Omron CX-Programmer project 新工程 (CX-Programmer 5.00)

# PLC 新PLC1: CQM1 CPU41

## Global symbols (name address type ; comment)
0.00 BOOL  ; 输送线全线启动
0.01 BOOL  ; 日运行停止
0.10 BOOL  ; 接触器KM1辅助触点
0.11 BOOL  ; 接触器KM2辅助触点
0.12 BOOL  ; 自动
0.13 BOOL  ; 手动
0.14 BOOL  ; 工位前占位
0.15 BOOL  ; 工位占位
100.00 BOOL  ; 输送电机M01-04接触器
100.01 BOOL  ; 输送电机M05-08接触器
100.02 BOOL  ; 输送电机M11-15接触器
100.05 BOOL  ; 输送电机M09接触器
100.06 BOOL  ; 输送电机M10接触器正转
100.07 BOOL  ; 输送电机M09接触器反转
100.10 BOOL  ; 1#密封试验开始
100.11 BOOL  ; 打号开始（接打号机）
100.12 BOOL  ; 输送线运行
101.03 BOOL  ; 自动指示灯
101.04 BOOL  ; 原位指示灯
101.05 BOOL  ; 自动指示灯
101.06 BOOL  ; 原位指示灯
101.07 BOOL  ; 自动指示灯
101.08 BOOL  ; 原位指示灯
103.00 BOOL  ; 工位前停止器
103.01 BOOL  ; 工位停止器
103.02 BOOL  ; 举升缸上升
103.03 BOOL  ; 上密封缸下降
103.04 BOOL  ; 上密封缸上升
103.05 BOOL  ; 左密封缸前进
103.06 BOOL  ; 左密封缸后退
103.07 BOOL  ; 排气孔密封缸前进
103.08 BOOL  ; 排气孔密封缸后退
103.10 BOOL  ; 2#密封试验开始
103.11 BOOL  ; 2#密封试验复位
103.12 BOOL  ; 举升缸下降
103.13 BOOL  ; 工位停止器
103.14 BOOL  ; 举升缸上升
103.15 BOOL  ; 上密封缸下降
104.00 BOOL  ; 上密封缸上升
104.01 BOOL  ; 左密封缸前进
104.02 BOOL  ; 左密封缸后退
104.03 BOOL  ; 排气孔密封缸前进
104.04 BOOL  ; 排气孔密封缸后退
104.06 BOOL  ; 工位停止器
104.07 BOOL  ; 举升缸上升
104.08 BOOL  ; 工位停止器（打号）
104.09 BOOL  ; 举升缸上升（打号）
104.10 BOOL  ; 举升缸下降（打号）
104.11 BOOL  ; 举升缸下降
104.12 BOOL  ; 举升缸下降
104.13 BOOL  ; 工位前停止器
150.02 BOOL  ; 输送线运行
160.00 BOOL  ; 自动
160.01 BOOL  ; 手动
160.03 BOOL  ; 密封机原状态
160.05 BOOL  ; 试验确认
160.07 BOOL  ; 试验不合格
160.08 BOOL  ; 试验合格
160.10 BOOL  ; 检测无工件确认
161.00 BOOL  ; 自动
161.01 BOOL  ; 手动
161.03 BOOL  ; 密封机原状态
161.05 BOOL  ; 试验确认
161.07 BOOL  ; 试验不合格
161.08 BOOL  ; 试验合格
161.10 BOOL  ; 检测无工件确认
162.00 BOOL  ; 工位前停止器
162.01 BOOL  ; 举升缸上升
162.02 BOOL  ; 举升缸下降
162.03 BOOL  ; 上密封缸下降
162.04 BOOL  ; 上密封缸上升
162.05 BOOL  ; 左密封缸前进
162.06 BOOL  ; 左密封缸后退
162.07 BOOL  ; 排气孔密封缸前进
162.08 BOOL  ; 排气孔密封缸后退
162.09 BOOL  ; 工位停止器
162.11 BOOL  ; 密封试验开始
162.14 BOOL  ; 使162.11失电
163.00 BOOL  ; 工位前停止器
163.01 BOOL  ; 举升缸上升
163.02 BOOL  ; 举升缸下降
163.03 BOOL  ; 上密封缸下降
163.04 BOOL  ; 上密封缸上升
163.05 BOOL  ; 左密封缸前进
163.06 BOOL  ; 左密封缸后退
163.07 BOOL  ; 排气孔密封缸前进
163.08 BOOL  ; 排气孔密封缸后退
163.09 BOOL  ; 工位停止器
163.11 BOOL  ; 密封试验开始
163.14 BOOL  ; 使163.11失电
170.00 BOOL  ; 自动
170.01 BOOL  ; 手动
170.03 BOOL  ; 举升缸下位
170.04 BOOL  ; 举升缸下位（打号）
172.01 BOOL  ; 举升缸上升
172.02 BOOL  ; 举升缸下降
172.05 BOOL  ; 电机M10正转
172.06 BOOL  ; 电机M09反转
172.08 BOOL  ; 工位停止器
172.10 BOOL  ; 举升缸上升（打号）
172.11 BOOL  ; 举升缸下降（打号）
172.12 BOOL  ; 工位停止器（打号）
172.13 BOOL  ; 打号开始
1.01 BOOL  ; 有无工件检测
1.02 BOOL  ; 变速箱类型检测
1.04 BOOL  ; 举升缸下位
1.05 BOOL  ; 举升缸上位
1.06 BOOL  ; 上密封缸上位
1.07 BOOL  ; 上密封缸下位
1.08 BOOL  ; 左密封缸后位
1.09 BOOL  ; 左密封缸前位
1.12 BOOL  ; 排气孔密封缸后位
1.13 BOOL  ; 排气孔密封缸前位
1.15 BOOL  ; 品种选择
2.00 BOOL  ; 试验合格
2.01 BOOL  ; 试验不合格
2.02 BOOL  ; 工件放行确认
2.04 BOOL  ; 举升缸上升
2.05 BOOL  ; 举升缸下降
2.06 BOOL  ; 上密封缸下降
2.07 BOOL  ; 上密封缸上升
2.08 BOOL  ; 左密封缸向前
2.09 BOOL  ; 左密封缸向后
2.10 BOOL  ; 排气孔密封缸向前
2.11 BOOL  ; 排气孔密封缸向后
2.12 BOOL  ; 标记缸动作
2.13 BOOL  ; 工位前停止器下
2.14 BOOL  ; 工位停止器下
2.15 BOOL  ; 信号灯测试
3.00 BOOL  ; 工件进维修段确认
3.01 BOOL  ; 自动
3.02 BOOL  ; 手动
3.03 BOOL  ; 工位占位
3.04 BOOL  ; 有无工件检测
3.05 BOOL  ; 举升缸下位
3.06 BOOL  ; 举升缸上位
3.07 BOOL  ; 上密封缸上位
3.08 BOOL  ; 上密封缸下位
3.09 BOOL  ; 左密封缸后位
3.10 BOOL  ; 左密封缸前位
3.11 BOOL  ; 排气孔密封缸后位
3.12 BOOL  ; 排气孔密封缸前位
3.13 BOOL  ; 工位前占位
3.14 BOOL  ; 试验合格
3.15 BOOL  ; 试验不合格
4.01 BOOL  ; 举升缸上升
4.02 BOOL  ; 举升缸下降
4.03 BOOL  ; 上密封缸下降
4.04 BOOL  ; 上密封缸上升
4.05 BOOL  ; 左密封缸向前
4.06 BOOL  ; 左密封缸向后
4.07 BOOL  ; 排气孔密封缸向前
4.08 BOOL  ; 排气孔密封缸向后
4.09 BOOL  ; 工位停止器下
4.10 BOOL  ; 信号灯测试
4.11 BOOL  ; 工件放行确认
4.12 BOOL  ; 工位前停止器下
4.13 BOOL  ; 预留（暂未用）
4.14 BOOL  ; 自动
4.15 BOOL  ; 手动
5.00 BOOL  ; 工位托盘占位
5.01 BOOL  ; 举升缸下位
5.02 BOOL  ; 举升缸上位
5.03 BOOL  ; 转移前到位
5.04 BOOL  ; 转移后到位
5.07 BOOL  ; 工位托盘占位（打号）
5.08 BOOL  ; 托盘满位（打号）
5.09 BOOL  ; 举升缸下位（打号）
5.10 BOOL  ; 举升缸上位（打号）
5.11 BOOL  ; 打号完毕（打号）
5.14 BOOL  ; 举升缸上升
5.15 BOOL  ; 举升缸下降
6.00 BOOL  ; 转移向前（+打号）
6.01 BOOL  ; 转移向后（+打号）
6.02 BOOL  ; 维修段放行（+打号）
6.03 BOOL  ; 出维修段确认（+打号）
6.04 BOOL  ; 打号工位举升（+打号）
6.05 BOOL  ; 打号工位下降（+打号）
6.06 BOOL  ; 打号工位放行（+打号）
6.07 BOOL  ; 信号灯测试（+打号）

## Program 新程序1 (no task)

### Section 段1_启动

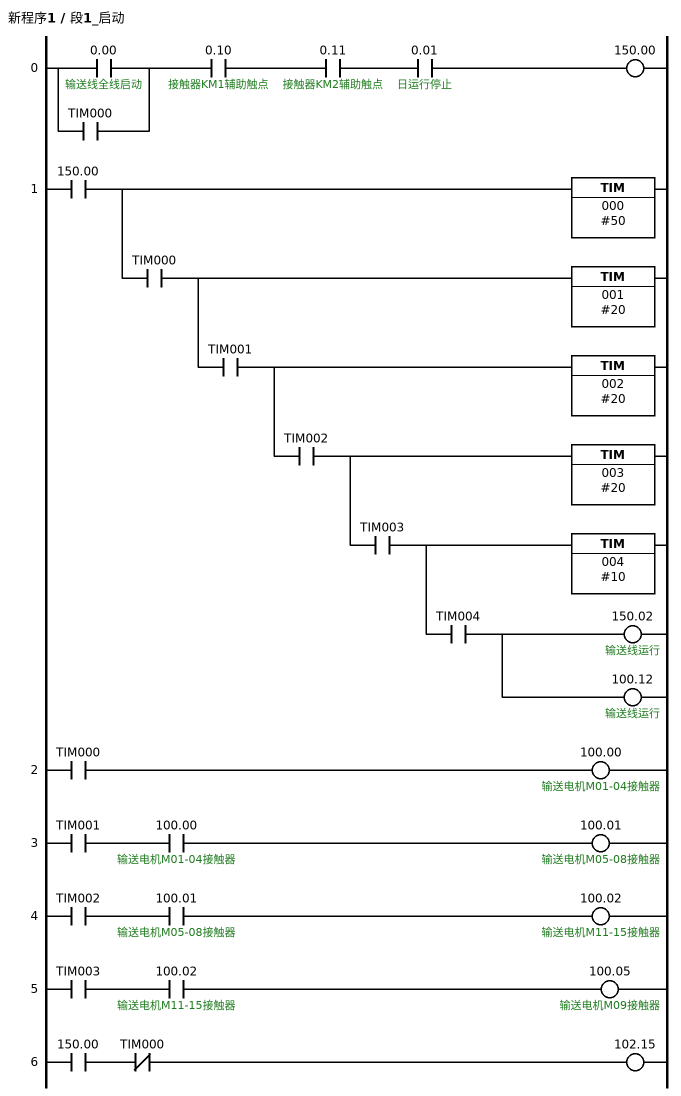
; rung 0
LD 0.00  ; 输送线全线启动
OR TIM000
AND 0.10  ; 接触器KM1辅助触点
AND 0.11  ; 接触器KM2辅助触点
AND 0.01  ; 日运行停止
OUT 150.00
; rung 1
LD 150.00
TIM 000 #50
AND TIM000
TIM 001 #20
AND TIM001
TIM 002 #20
AND TIM002
TIM 003 #20
AND TIM003
TIM 004 #10
AND TIM004
OUT 150.02  ; 输送线运行
OUT 100.12  ; 输送线运行
; rung 2
LD TIM000
OUT 100.00  ; 输送电机M01-04接触器
; rung 3
LD TIM001
AND 100.00  ; 输送电机M01-04接触器
OUT 100.01  ; 输送电机M05-08接触器
; rung 4
LD TIM002
AND 100.01  ; 输送电机M05-08接触器
OUT 100.02  ; 输送电机M11-15接触器
; rung 5
LD TIM003
AND 100.02  ; 输送电机M11-15接触器
OUT 100.05  ; 输送电机M09接触器
; rung 6
LD 150.00
ANDNOT TIM000
OUT 102.15

### Section 段2_试验机1

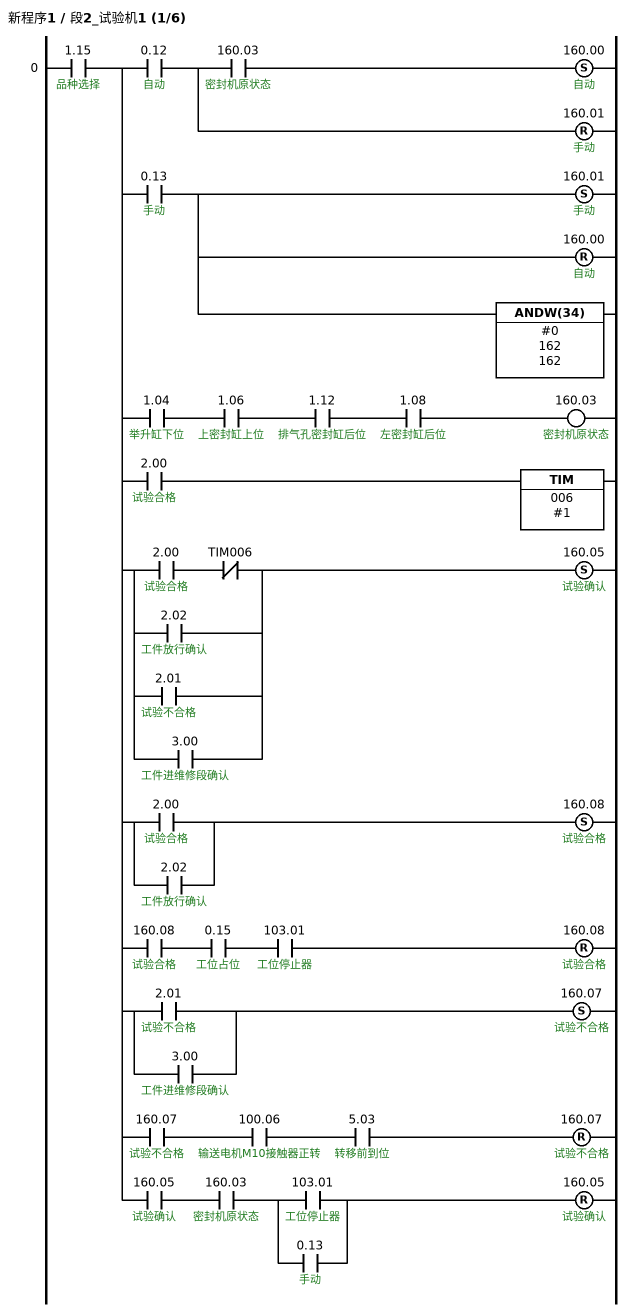
; rung 0
LD 1.15  ; 品种选择
OUT TR0
AND 0.12  ; 自动
OUT TR1
AND 160.03  ; 密封机原状态
SET 160.00  ; 自动
LD TR1
RSET 160.01  ; 手动
LD TR0
AND 0.13  ; 手动
SET 160.01  ; 手动
RSET 160.00  ; 自动
ANDW(34) #0 162 162
LD TR0
AND 1.04  ; 举升缸下位
AND 1.06  ; 上密封缸上位
AND 1.12  ; 排气孔密封缸后位
AND 1.08  ; 左密封缸后位
OUT 160.03  ; 密封机原状态
LD TR0
AND 2.00  ; 试验合格
TIM 006 #1
LD TR0
LD 2.00  ; 试验合格
ANDNOT TIM006
OR 2.02  ; 工件放行确认
OR 2.01  ; 试验不合格
OR 3.00  ; 工件进维修段确认
ANDLD
SET 160.05  ; 试验确认
LD TR0
LD 2.00  ; 试验合格
OR 2.02  ; 工件放行确认
ANDLD
SET 160.08  ; 试验合格
LD TR0
AND 160.08  ; 试验合格
AND 0.15  ; 工位占位
AND 103.01  ; 工位停止器
RSET 160.08  ; 试验合格
LD TR0
LD 2.01  ; 试验不合格
OR 3.00  ; 工件进维修段确认
ANDLD
SET 160.07  ; 试验不合格
LD TR0
AND 160.07  ; 试验不合格
AND 100.06  ; 输送电机M10接触器正转
AND 5.03  ; 转移前到位
RSET 160.07  ; 试验不合格
LD TR0
AND 160.05  ; 试验确认
AND 160.03  ; 密封机原状态
LD 103.01  ; 工位停止器
OR 0.13  ; 手动
ANDLD
RSET 160.05  ; 试验确认

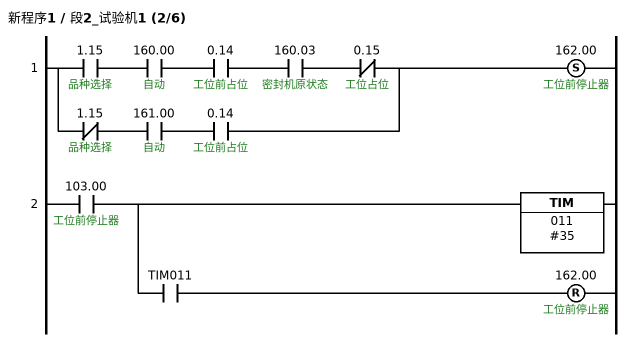
; rung 1
LD 1.15  ; 品种选择
AND 160.00  ; 自动
AND 0.14  ; 工位前占位
AND 160.03  ; 密封机原状态
ANDNOT 0.15  ; 工位占位
LDNOT 1.15  ; 品种选择
AND 161.00  ; 自动
AND 0.14  ; 工位前占位
ORLD
SET 162.00  ; 工位前停止器
; rung 2
LD 103.00  ; 工位前停止器
TIM 011 #35
AND TIM011
RSET 162.00  ; 工位前停止器

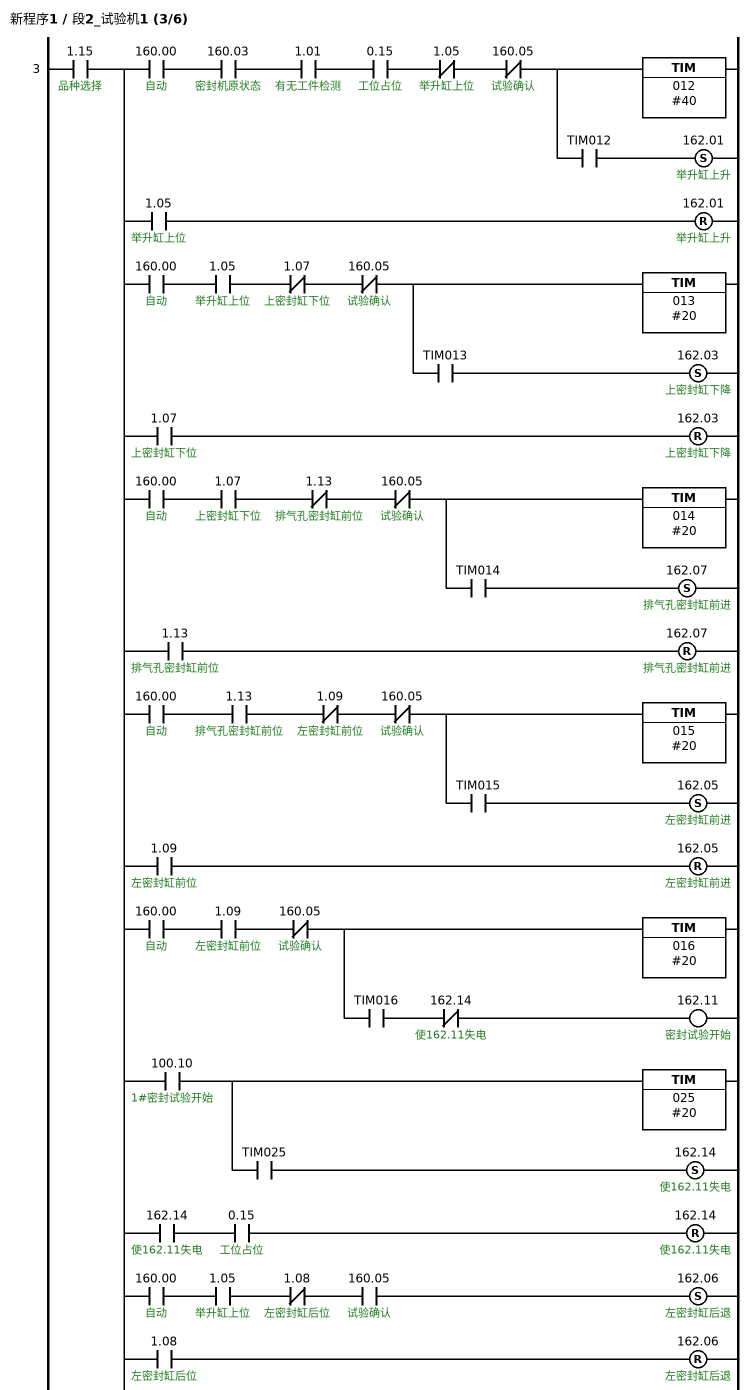

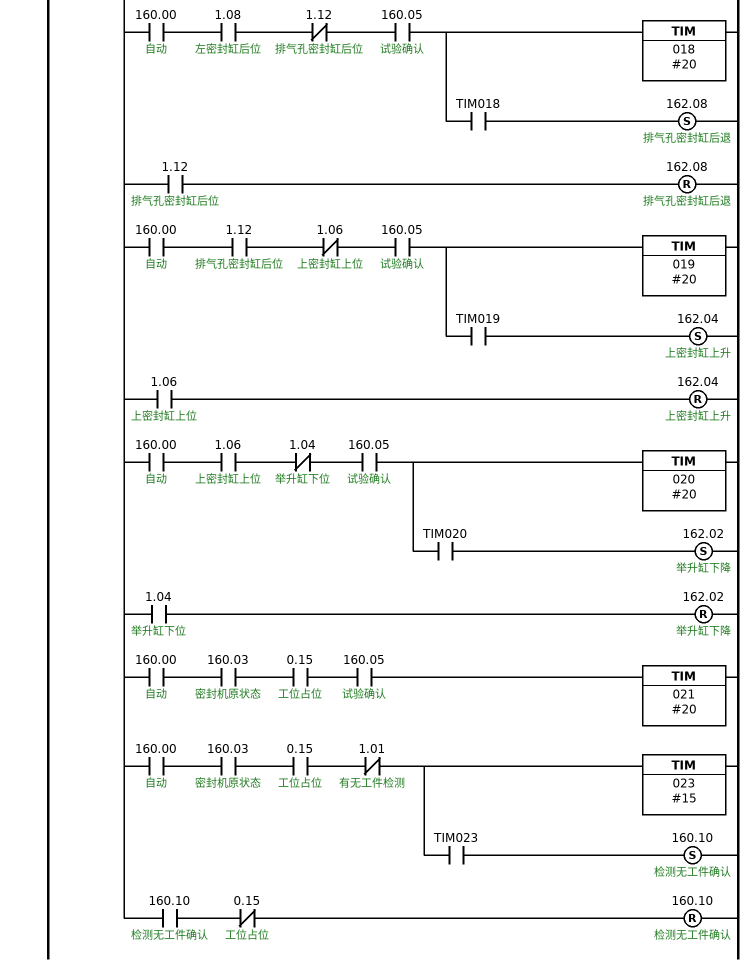
; rung 3
LD 1.15  ; 品种选择
OUT TR0
AND 160.00  ; 自动
AND 160.03  ; 密封机原状态
AND 1.01  ; 有无工件检测
AND 0.15  ; 工位占位
ANDNOT 1.05  ; 举升缸上位
ANDNOT 160.05  ; 试验确认
TIM 012 #40
AND TIM012
SET 162.01  ; 举升缸上升
LD TR0
AND 1.05  ; 举升缸上位
RSET 162.01  ; 举升缸上升
LD TR0
AND 160.00  ; 自动
AND 1.05  ; 举升缸上位
ANDNOT 1.07  ; 上密封缸下位
ANDNOT 160.05  ; 试验确认
TIM 013 #20
AND TIM013
SET 162.03  ; 上密封缸下降
LD TR0
AND 1.07  ; 上密封缸下位
RSET 162.03  ; 上密封缸下降
LD TR0
AND 160.00  ; 自动
AND 1.07  ; 上密封缸下位
ANDNOT 1.13  ; 排气孔密封缸前位
ANDNOT 160.05  ; 试验确认
TIM 014 #20
AND TIM014
SET 162.07  ; 排气孔密封缸前进
LD TR0
AND 1.13  ; 排气孔密封缸前位
RSET 162.07  ; 排气孔密封缸前进
LD TR0
AND 160.00  ; 自动
AND 1.13  ; 排气孔密封缸前位
ANDNOT 1.09  ; 左密封缸前位
ANDNOT 160.05  ; 试验确认
TIM 015 #20
AND TIM015
SET 162.05  ; 左密封缸前进
LD TR0
AND 1.09  ; 左密封缸前位
RSET 162.05  ; 左密封缸前进
LD TR0
AND 160.00  ; 自动
AND 1.09  ; 左密封缸前位
ANDNOT 160.05  ; 试验确认
TIM 016 #20
AND TIM016
ANDNOT 162.14  ; 使162.11失电
OUT 162.11  ; 密封试验开始
LD TR0
AND 100.10  ; 1#密封试验开始
TIM 025 #20
AND TIM025
SET 162.14  ; 使162.11失电
LD TR0
AND 162.14  ; 使162.11失电
AND 0.15  ; 工位占位
RSET 162.14  ; 使162.11失电
LD TR0
AND 160.00  ; 自动
AND 1.05  ; 举升缸上位
ANDNOT 1.08  ; 左密封缸后位
AND 160.05  ; 试验确认
SET 162.06  ; 左密封缸后退
LD TR0
AND 1.08  ; 左密封缸后位
RSET 162.06  ; 左密封缸后退
LD TR0
AND 160.00  ; 自动
AND 1.08  ; 左密封缸后位
ANDNOT 1.12  ; 排气孔密封缸后位
AND 160.05  ; 试验确认
TIM 018 #20
AND TIM018
SET 162.08  ; 排气孔密封缸后退
LD TR0
AND 1.12  ; 排气孔密封缸后位
RSET 162.08  ; 排气孔密封缸后退
LD TR0
AND 160.00  ; 自动
AND 1.12  ; 排气孔密封缸后位
ANDNOT 1.06  ; 上密封缸上位
AND 160.05  ; 试验确认
TIM 019 #20
AND TIM019
SET 162.04  ; 上密封缸上升
LD TR0
AND 1.06  ; 上密封缸上位
RSET 162.04  ; 上密封缸上升
LD TR0
AND 160.00  ; 自动
AND 1.06  ; 上密封缸上位
ANDNOT 1.04  ; 举升缸下位
AND 160.05  ; 试验确认
TIM 020 #20
AND TIM020
SET 162.02  ; 举升缸下降
LD TR0
AND 1.04  ; 举升缸下位
RSET 162.02  ; 举升缸下降
LD TR0
AND 160.00  ; 自动
AND 160.03  ; 密封机原状态
AND 0.15  ; 工位占位
AND 160.05  ; 试验确认
TIM 021 #20
LD TR0
AND 160.00  ; 自动
AND 160.03  ; 密封机原状态
AND 0.15  ; 工位占位
ANDNOT 1.01  ; 有无工件检测
TIM 023 #15
AND TIM023
SET 160.10  ; 检测无工件确认
LD TR0
AND 160.10  ; 检测无工件确认
ANDNOT 0.15  ; 工位占位
RSET 160.10  ; 检测无工件确认

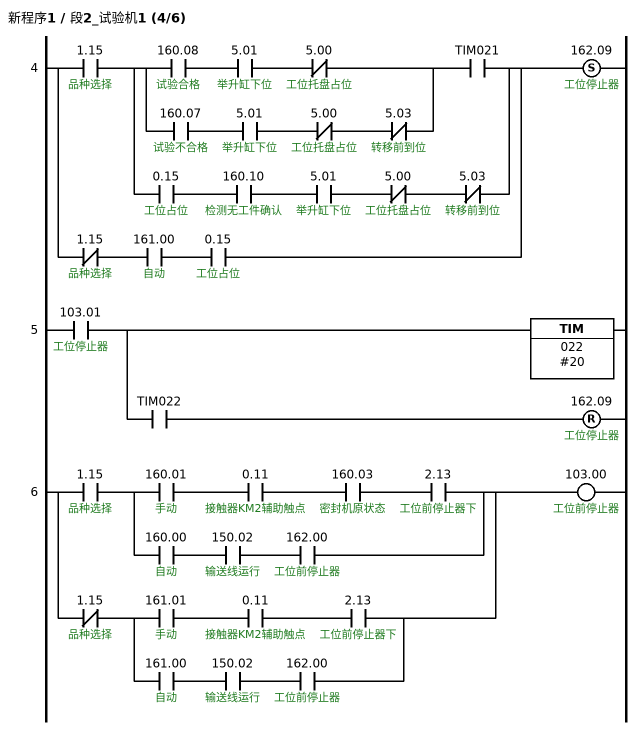
; rung 4
LD 1.15  ; 品种选择
LD 160.08  ; 试验合格
AND 5.01  ; 举升缸下位
ANDNOT 5.00  ; 工位托盘占位
LD 160.07  ; 试验不合格
AND 5.01  ; 举升缸下位
ANDNOT 5.00  ; 工位托盘占位
ANDNOT 5.03  ; 转移前到位
ORLD
AND TIM021
LD 0.15  ; 工位占位
AND 160.10  ; 检测无工件确认
AND 5.01  ; 举升缸下位
ANDNOT 5.00  ; 工位托盘占位
ANDNOT 5.03  ; 转移前到位
ORLD
ANDLD
LDNOT 1.15  ; 品种选择
AND 161.00  ; 自动
AND 0.15  ; 工位占位
ORLD
SET 162.09  ; 工位停止器
; rung 5
LD 103.01  ; 工位停止器
TIM 022 #20
AND TIM022
RSET 162.09  ; 工位停止器
; rung 6
LD 1.15  ; 品种选择
LD 160.01  ; 手动
AND 0.11  ; 接触器KM2辅助触点
AND 160.03  ; 密封机原状态
AND 2.13  ; 工位前停止器下
LD 160.00  ; 自动
AND 150.02  ; 输送线运行
AND 162.00  ; 工位前停止器
ORLD
ANDLD
LDNOT 1.15  ; 品种选择
LD 161.01  ; 手动
AND 0.11  ; 接触器KM2辅助触点
AND 2.13  ; 工位前停止器下
LD 161.00  ; 自动
AND 150.02  ; 输送线运行
AND 162.00  ; 工位前停止器
ORLD
ANDLD
ORLD
OUT 103.00  ; 工位前停止器

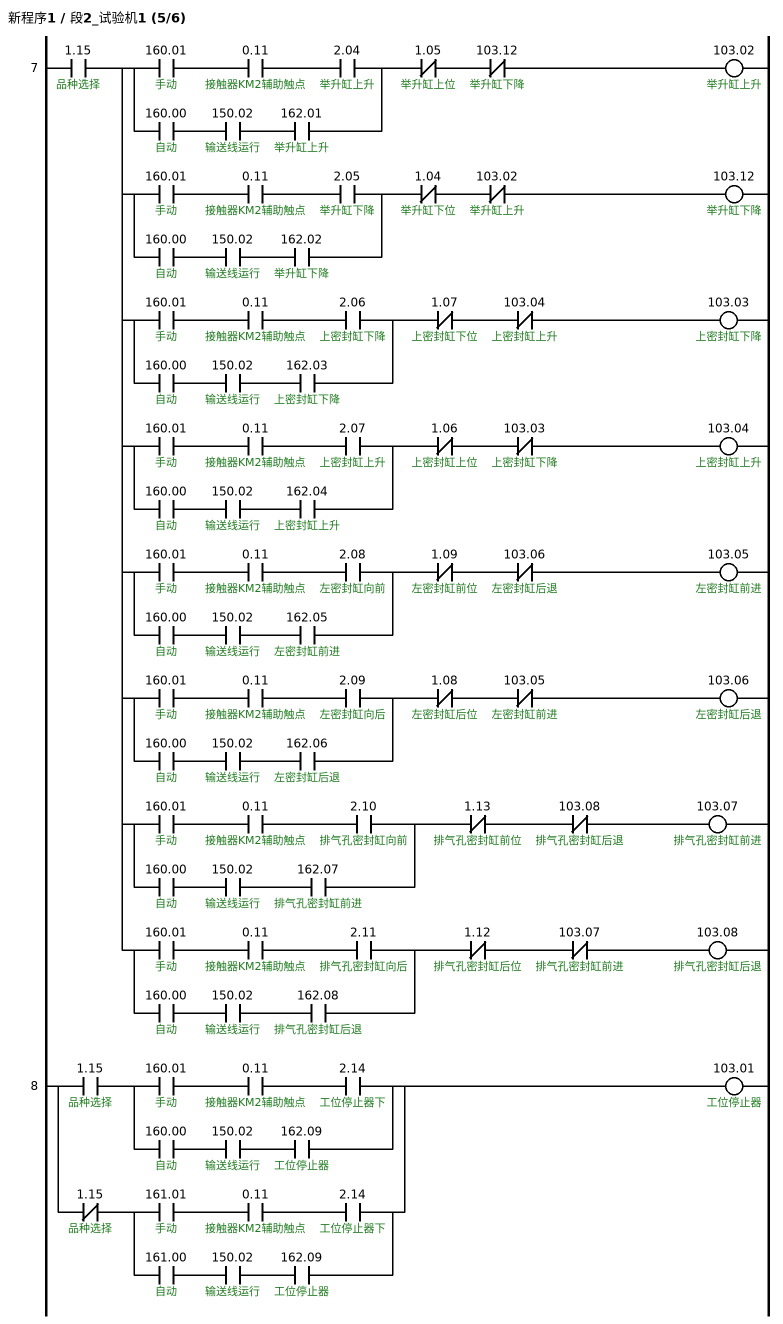
; rung 7
LD 1.15  ; 品种选择
OUT TR0
LD 160.01  ; 手动
AND 0.11  ; 接触器KM2辅助触点
AND 2.04  ; 举升缸上升
LD 160.00  ; 自动
AND 150.02  ; 输送线运行
AND 162.01  ; 举升缸上升
ORLD
ANDLD
ANDNOT 1.05  ; 举升缸上位
ANDNOT 103.12  ; 举升缸下降
OUT 103.02  ; 举升缸上升
LD TR0
LD 160.01  ; 手动
AND 0.11  ; 接触器KM2辅助触点
AND 2.05  ; 举升缸下降
LD 160.00  ; 自动
AND 150.02  ; 输送线运行
AND 162.02  ; 举升缸下降
ORLD
ANDLD
ANDNOT 1.04  ; 举升缸下位
ANDNOT 103.02  ; 举升缸上升
OUT 103.12  ; 举升缸下降
LD TR0
LD 160.01  ; 手动
AND 0.11  ; 接触器KM2辅助触点
AND 2.06  ; 上密封缸下降
LD 160.00  ; 自动
AND 150.02  ; 输送线运行
AND 162.03  ; 上密封缸下降
ORLD
ANDLD
ANDNOT 1.07  ; 上密封缸下位
ANDNOT 103.04  ; 上密封缸上升
OUT 103.03  ; 上密封缸下降
LD TR0
LD 160.01  ; 手动
AND 0.11  ; 接触器KM2辅助触点
AND 2.07  ; 上密封缸上升
LD 160.00  ; 自动
AND 150.02  ; 输送线运行
AND 162.04  ; 上密封缸上升
ORLD
ANDLD
ANDNOT 1.06  ; 上密封缸上位
ANDNOT 103.03  ; 上密封缸下降
OUT 103.04  ; 上密封缸上升
LD TR0
LD 160.01  ; 手动
AND 0.11  ; 接触器KM2辅助触点
AND 2.08  ; 左密封缸向前
LD 160.00  ; 自动
AND 150.02  ; 输送线运行
AND 162.05  ; 左密封缸前进
ORLD
ANDLD
ANDNOT 1.09  ; 左密封缸前位
ANDNOT 103.06  ; 左密封缸后退
OUT 103.05  ; 左密封缸前进
LD TR0
LD 160.01  ; 手动
AND 0.11  ; 接触器KM2辅助触点
AND 2.09  ; 左密封缸向后
LD 160.00  ; 自动
AND 150.02  ; 输送线运行
AND 162.06  ; 左密封缸后退
ORLD
ANDLD
ANDNOT 1.08  ; 左密封缸后位
ANDNOT 103.05  ; 左密封缸前进
OUT 103.06  ; 左密封缸后退
LD TR0
LD 160.01  ; 手动
AND 0.11  ; 接触器KM2辅助触点
AND 2.10  ; 排气孔密封缸向前
LD 160.00  ; 自动
AND 150.02  ; 输送线运行
AND 162.07  ; 排气孔密封缸前进
ORLD
ANDLD
ANDNOT 1.13  ; 排气孔密封缸前位
ANDNOT 103.08  ; 排气孔密封缸后退
OUT 103.07  ; 排气孔密封缸前进
LD TR0
LD 160.01  ; 手动
AND 0.11  ; 接触器KM2辅助触点
AND 2.11  ; 排气孔密封缸向后
LD 160.00  ; 自动
AND 150.02  ; 输送线运行
AND 162.08  ; 排气孔密封缸后退
ORLD
ANDLD
ANDNOT 1.12  ; 排气孔密封缸后位
ANDNOT 103.07  ; 排气孔密封缸前进
OUT 103.08  ; 排气孔密封缸后退
; rung 8
LD 1.15  ; 品种选择
LD 160.01  ; 手动
AND 0.11  ; 接触器KM2辅助触点
AND 2.14  ; 工位停止器下
LD 160.00  ; 自动
AND 150.02  ; 输送线运行
AND 162.09  ; 工位停止器
ORLD
ANDLD
LDNOT 1.15  ; 品种选择
LD 161.01  ; 手动
AND 0.11  ; 接触器KM2辅助触点
AND 2.14  ; 工位停止器下
LD 161.00  ; 自动
AND 150.02  ; 输送线运行
AND 162.09  ; 工位停止器
ORLD
ANDLD
ORLD
OUT 103.01  ; 工位停止器

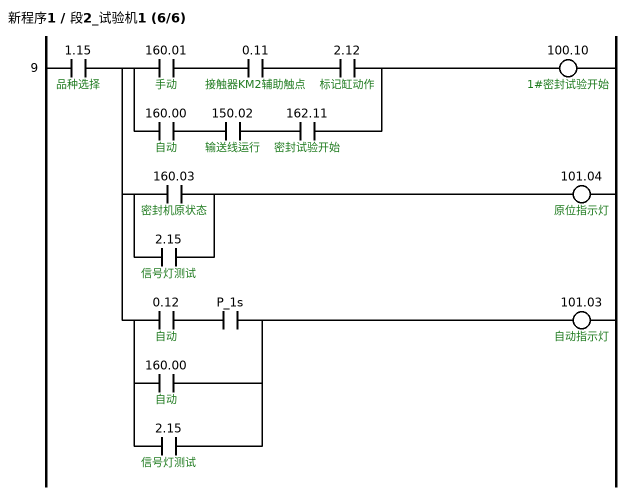
; rung 9
LD 1.15  ; 品种选择
OUT TR0
LD 160.01  ; 手动
AND 0.11  ; 接触器KM2辅助触点
AND 2.12  ; 标记缸动作
LD 160.00  ; 自动
AND 150.02  ; 输送线运行
AND 162.11  ; 密封试验开始
ORLD
ANDLD
OUT 100.10  ; 1#密封试验开始
LD TR0
LD 160.03  ; 密封机原状态
OR 2.15  ; 信号灯测试
ANDLD
OUT 101.04  ; 原位指示灯
LD TR0
LD 0.12  ; 自动
AND P_1s
OR 160.00  ; 自动
OR 2.15  ; 信号灯测试
ANDLD
OUT 101.03  ; 自动指示灯

### Section 段3_试验机2

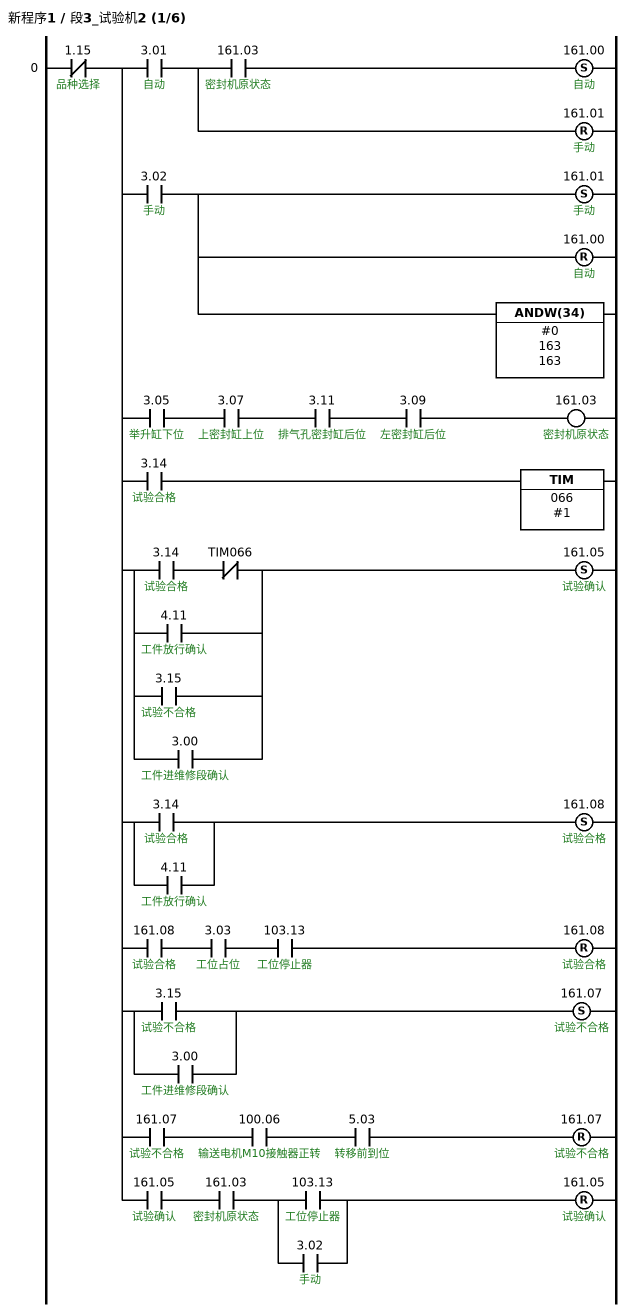
; rung 0
LDNOT 1.15  ; 品种选择
OUT TR0
AND 3.01  ; 自动
OUT TR1
AND 161.03  ; 密封机原状态
SET 161.00  ; 自动
LD TR1
RSET 161.01  ; 手动
LD TR0
AND 3.02  ; 手动
SET 161.01  ; 手动
RSET 161.00  ; 自动
ANDW(34) #0 163 163
LD TR0
AND 3.05  ; 举升缸下位
AND 3.07  ; 上密封缸上位
AND 3.11  ; 排气孔密封缸后位
AND 3.09  ; 左密封缸后位
OUT 161.03  ; 密封机原状态
LD TR0
AND 3.14  ; 试验合格
TIM 066 #1
LD TR0
LD 3.14  ; 试验合格
ANDNOT TIM066
OR 4.11  ; 工件放行确认
OR 3.15  ; 试验不合格
OR 3.00  ; 工件进维修段确认
ANDLD
SET 161.05  ; 试验确认
LD TR0
LD 3.14  ; 试验合格
OR 4.11  ; 工件放行确认
ANDLD
SET 161.08  ; 试验合格
LD TR0
AND 161.08  ; 试验合格
AND 3.03  ; 工位占位
AND 103.13  ; 工位停止器
RSET 161.08  ; 试验合格
LD TR0
LD 3.15  ; 试验不合格
OR 3.00  ; 工件进维修段确认
ANDLD
SET 161.07  ; 试验不合格
LD TR0
AND 161.07  ; 试验不合格
AND 100.06  ; 输送电机M10接触器正转
AND 5.03  ; 转移前到位
RSET 161.07  ; 试验不合格
LD TR0
AND 161.05  ; 试验确认
AND 161.03  ; 密封机原状态
LD 103.13  ; 工位停止器
OR 3.02  ; 手动
ANDLD
RSET 161.05  ; 试验确认

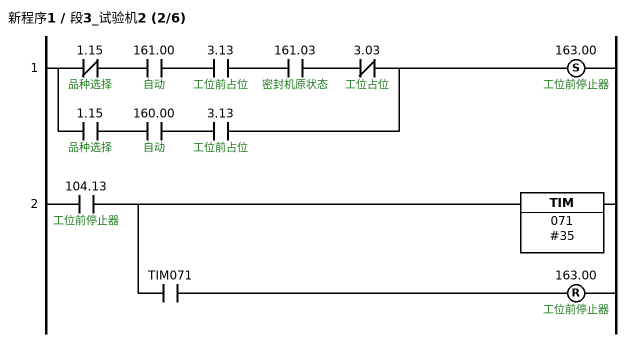
; rung 1
LDNOT 1.15  ; 品种选择
AND 161.00  ; 自动
AND 3.13  ; 工位前占位
AND 161.03  ; 密封机原状态
ANDNOT 3.03  ; 工位占位
LD 1.15  ; 品种选择
AND 160.00  ; 自动
AND 3.13  ; 工位前占位
ORLD
SET 163.00  ; 工位前停止器
; rung 2
LD 104.13  ; 工位前停止器
TIM 071 #35
AND TIM071
RSET 163.00  ; 工位前停止器

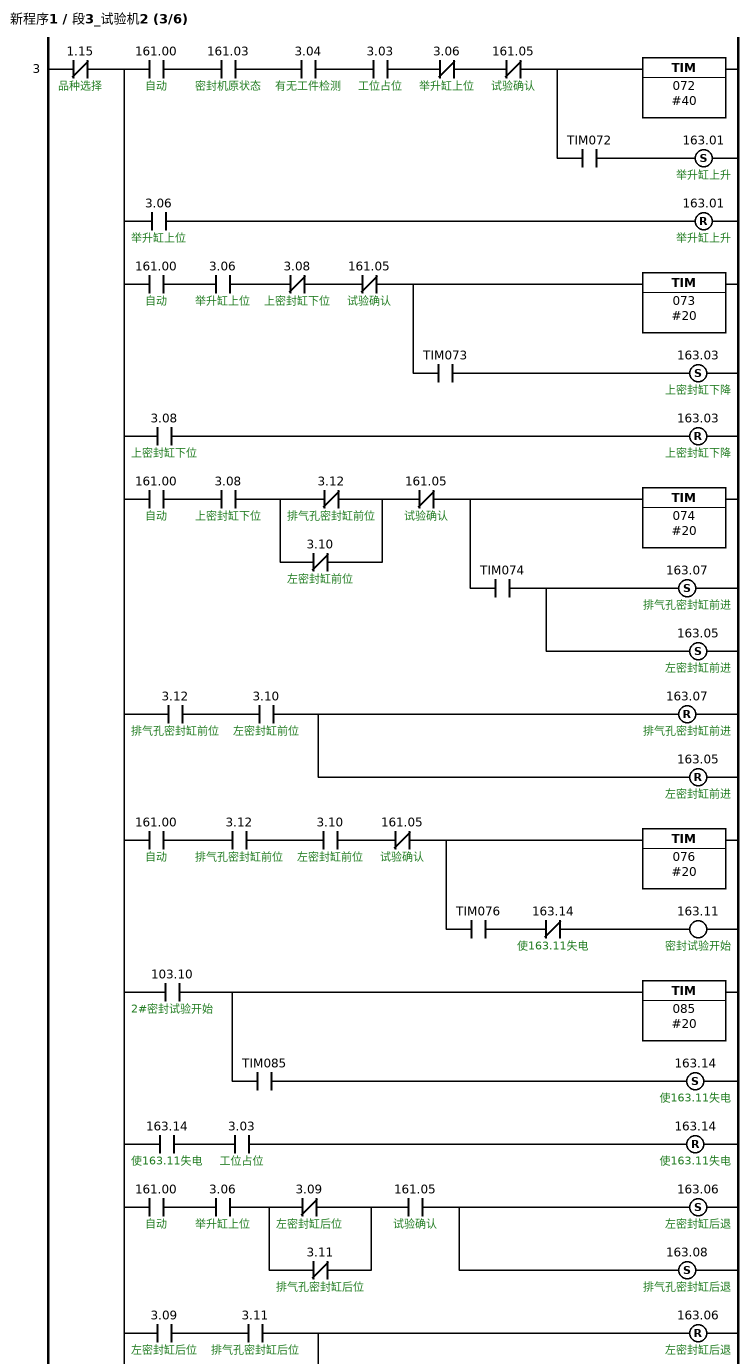

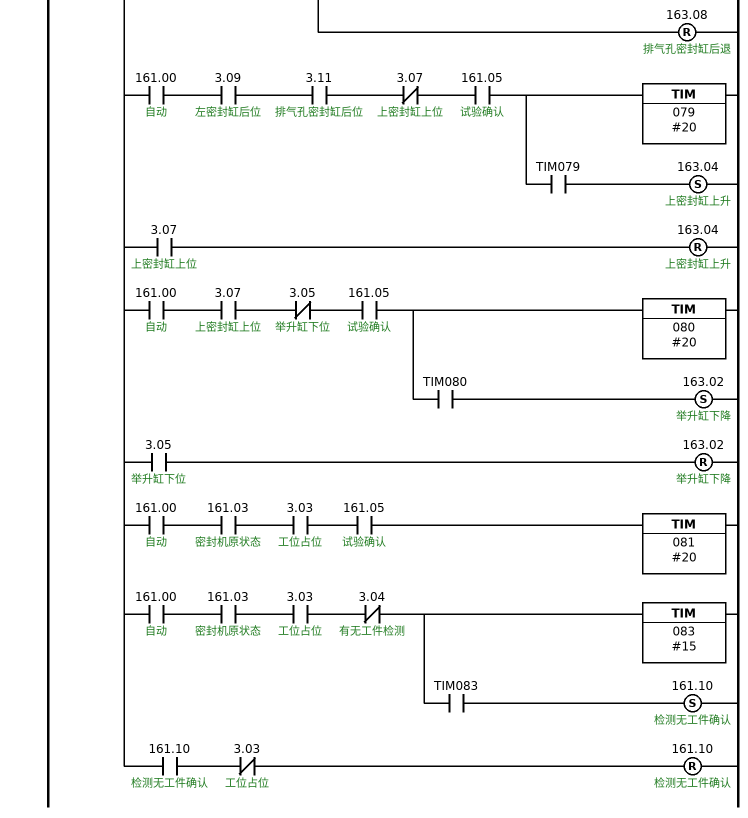
; rung 3
LDNOT 1.15  ; 品种选择
OUT TR0
AND 161.00  ; 自动
AND 161.03  ; 密封机原状态
AND 3.04  ; 有无工件检测
AND 3.03  ; 工位占位
ANDNOT 3.06  ; 举升缸上位
ANDNOT 161.05  ; 试验确认
TIM 072 #40
AND TIM072
SET 163.01  ; 举升缸上升
LD TR0
AND 3.06  ; 举升缸上位
RSET 163.01  ; 举升缸上升
LD TR0
AND 161.00  ; 自动
AND 3.06  ; 举升缸上位
ANDNOT 3.08  ; 上密封缸下位
ANDNOT 161.05  ; 试验确认
TIM 073 #20
AND TIM073
SET 163.03  ; 上密封缸下降
LD TR0
AND 3.08  ; 上密封缸下位
RSET 163.03  ; 上密封缸下降
LD TR0
AND 161.00  ; 自动
AND 3.08  ; 上密封缸下位
LDNOT 3.12  ; 排气孔密封缸前位
ORNOT 3.10  ; 左密封缸前位
ANDLD
ANDNOT 161.05  ; 试验确认
TIM 074 #20
AND TIM074
SET 163.07  ; 排气孔密封缸前进
SET 163.05  ; 左密封缸前进
LD TR0
AND 3.12  ; 排气孔密封缸前位
AND 3.10  ; 左密封缸前位
RSET 163.07  ; 排气孔密封缸前进
RSET 163.05  ; 左密封缸前进
LD TR0
AND 161.00  ; 自动
AND 3.12  ; 排气孔密封缸前位
AND 3.10  ; 左密封缸前位
ANDNOT 161.05  ; 试验确认
TIM 076 #20
AND TIM076
ANDNOT 163.14  ; 使163.11失电
OUT 163.11  ; 密封试验开始
LD TR0
AND 103.10  ; 2#密封试验开始
TIM 085 #20
AND TIM085
SET 163.14  ; 使163.11失电
LD TR0
AND 163.14  ; 使163.11失电
AND 3.03  ; 工位占位
RSET 163.14  ; 使163.11失电
LD TR0
AND 161.00  ; 自动
AND 3.06  ; 举升缸上位
LDNOT 3.09  ; 左密封缸后位
ORNOT 3.11  ; 排气孔密封缸后位
ANDLD
AND 161.05  ; 试验确认
SET 163.06  ; 左密封缸后退
SET 163.08  ; 排气孔密封缸后退
LD TR0
AND 3.09  ; 左密封缸后位
AND 3.11  ; 排气孔密封缸后位
RSET 163.06  ; 左密封缸后退
RSET 163.08  ; 排气孔密封缸后退
LD TR0
AND 161.00  ; 自动
AND 3.09  ; 左密封缸后位
AND 3.11  ; 排气孔密封缸后位
ANDNOT 3.07  ; 上密封缸上位
AND 161.05  ; 试验确认
TIM 079 #20
AND TIM079
SET 163.04  ; 上密封缸上升
LD TR0
AND 3.07  ; 上密封缸上位
RSET 163.04  ; 上密封缸上升
LD TR0
AND 161.00  ; 自动
AND 3.07  ; 上密封缸上位
ANDNOT 3.05  ; 举升缸下位
AND 161.05  ; 试验确认
TIM 080 #20
AND TIM080
SET 163.02  ; 举升缸下降
LD TR0
AND 3.05  ; 举升缸下位
RSET 163.02  ; 举升缸下降
LD TR0
AND 161.00  ; 自动
AND 161.03  ; 密封机原状态
AND 3.03  ; 工位占位
AND 161.05  ; 试验确认
TIM 081 #20
LD TR0
AND 161.00  ; 自动
AND 161.03  ; 密封机原状态
AND 3.03  ; 工位占位
ANDNOT 3.04  ; 有无工件检测
TIM 083 #15
AND TIM083
SET 161.10  ; 检测无工件确认
LD TR0
AND 161.10  ; 检测无工件确认
ANDNOT 3.03  ; 工位占位
RSET 161.10  ; 检测无工件确认

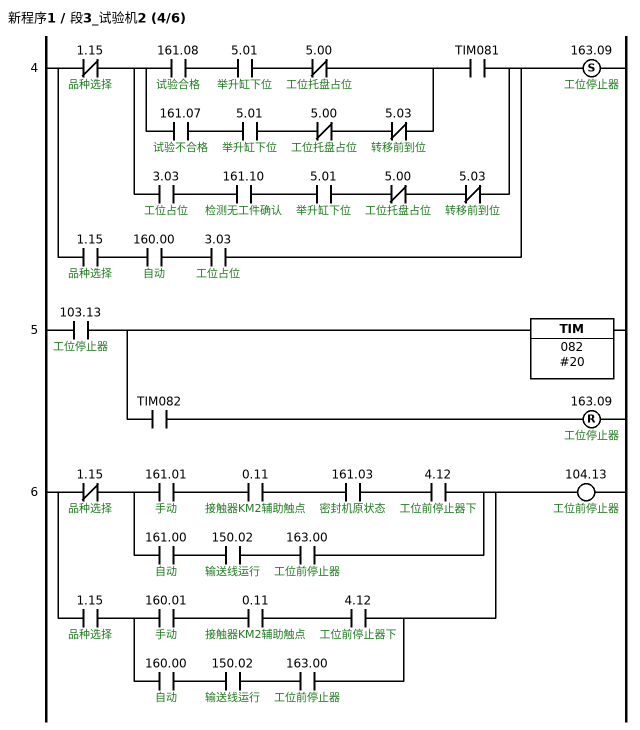
; rung 4
LDNOT 1.15  ; 品种选择
LD 161.08  ; 试验合格
AND 5.01  ; 举升缸下位
ANDNOT 5.00  ; 工位托盘占位
LD 161.07  ; 试验不合格
AND 5.01  ; 举升缸下位
ANDNOT 5.00  ; 工位托盘占位
ANDNOT 5.03  ; 转移前到位
ORLD
AND TIM081
LD 3.03  ; 工位占位
AND 161.10  ; 检测无工件确认
AND 5.01  ; 举升缸下位
ANDNOT 5.00  ; 工位托盘占位
ANDNOT 5.03  ; 转移前到位
ORLD
ANDLD
LD 1.15  ; 品种选择
AND 160.00  ; 自动
AND 3.03  ; 工位占位
ORLD
SET 163.09  ; 工位停止器
; rung 5
LD 103.13  ; 工位停止器
TIM 082 #20
AND TIM082
RSET 163.09  ; 工位停止器
; rung 6
LDNOT 1.15  ; 品种选择
LD 161.01  ; 手动
AND 0.11  ; 接触器KM2辅助触点
AND 161.03  ; 密封机原状态
AND 4.12  ; 工位前停止器下
LD 161.00  ; 自动
AND 150.02  ; 输送线运行
AND 163.00  ; 工位前停止器
ORLD
ANDLD
LD 1.15  ; 品种选择
LD 160.01  ; 手动
AND 0.11  ; 接触器KM2辅助触点
AND 4.12  ; 工位前停止器下
LD 160.00  ; 自动
AND 150.02  ; 输送线运行
AND 163.00  ; 工位前停止器
ORLD
ANDLD
ORLD
OUT 104.13  ; 工位前停止器

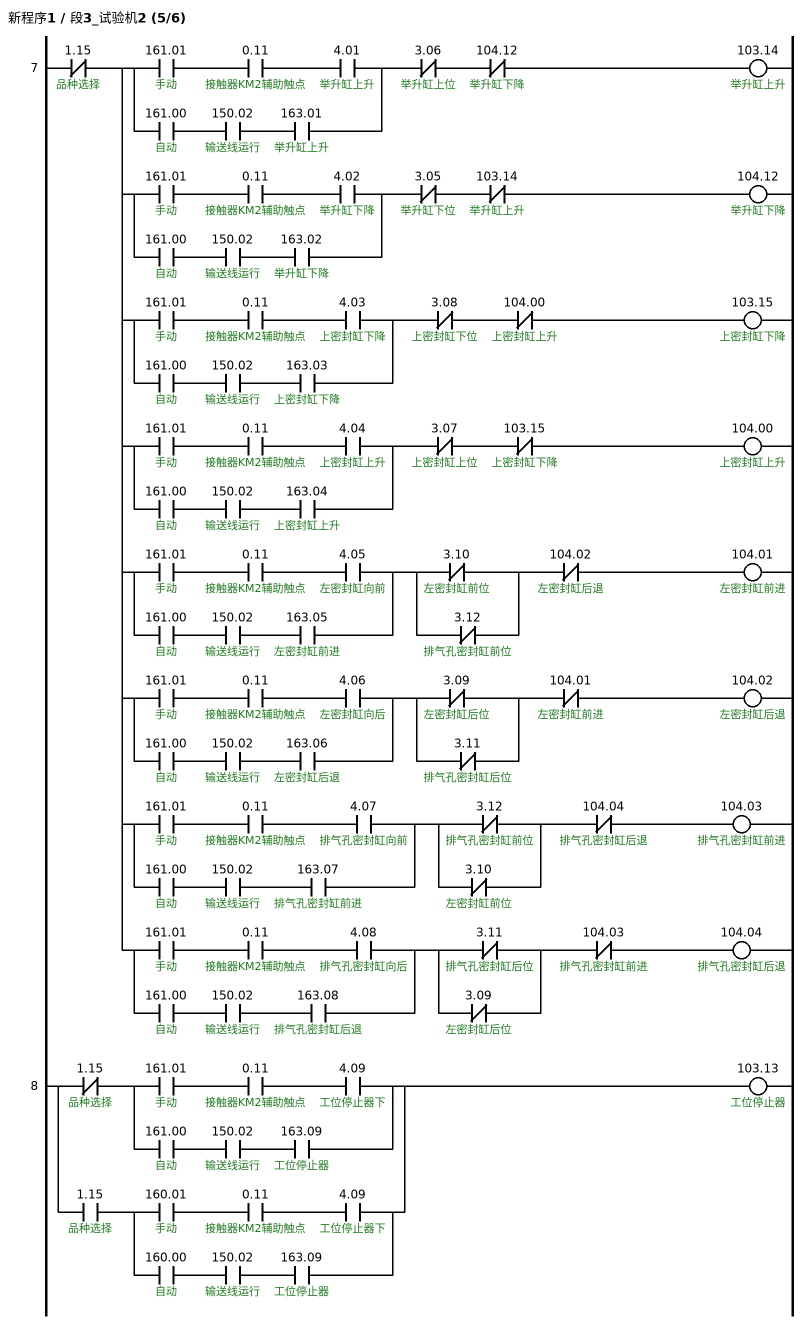
; rung 7
LDNOT 1.15  ; 品种选择
OUT TR0
LD 161.01  ; 手动
AND 0.11  ; 接触器KM2辅助触点
AND 4.01  ; 举升缸上升
LD 161.00  ; 自动
AND 150.02  ; 输送线运行
AND 163.01  ; 举升缸上升
ORLD
ANDLD
ANDNOT 3.06  ; 举升缸上位
ANDNOT 104.12  ; 举升缸下降
OUT 103.14  ; 举升缸上升
LD TR0
LD 161.01  ; 手动
AND 0.11  ; 接触器KM2辅助触点
AND 4.02  ; 举升缸下降
LD 161.00  ; 自动
AND 150.02  ; 输送线运行
AND 163.02  ; 举升缸下降
ORLD
ANDLD
ANDNOT 3.05  ; 举升缸下位
ANDNOT 103.14  ; 举升缸上升
OUT 104.12  ; 举升缸下降
LD TR0
LD 161.01  ; 手动
AND 0.11  ; 接触器KM2辅助触点
AND 4.03  ; 上密封缸下降
LD 161.00  ; 自动
AND 150.02  ; 输送线运行
AND 163.03  ; 上密封缸下降
ORLD
ANDLD
ANDNOT 3.08  ; 上密封缸下位
ANDNOT 104.00  ; 上密封缸上升
OUT 103.15  ; 上密封缸下降
LD TR0
LD 161.01  ; 手动
AND 0.11  ; 接触器KM2辅助触点
AND 4.04  ; 上密封缸上升
LD 161.00  ; 自动
AND 150.02  ; 输送线运行
AND 163.04  ; 上密封缸上升
ORLD
ANDLD
ANDNOT 3.07  ; 上密封缸上位
ANDNOT 103.15  ; 上密封缸下降
OUT 104.00  ; 上密封缸上升
LD TR0
LD 161.01  ; 手动
AND 0.11  ; 接触器KM2辅助触点
AND 4.05  ; 左密封缸向前
LD 161.00  ; 自动
AND 150.02  ; 输送线运行
AND 163.05  ; 左密封缸前进
ORLD
ANDLD
LDNOT 3.10  ; 左密封缸前位
ORNOT 3.12  ; 排气孔密封缸前位
ANDLD
ANDNOT 104.02  ; 左密封缸后退
OUT 104.01  ; 左密封缸前进
LD TR0
LD 161.01  ; 手动
AND 0.11  ; 接触器KM2辅助触点
AND 4.06  ; 左密封缸向后
LD 161.00  ; 自动
AND 150.02  ; 输送线运行
AND 163.06  ; 左密封缸后退
ORLD
ANDLD
LDNOT 3.09  ; 左密封缸后位
ORNOT 3.11  ; 排气孔密封缸后位
ANDLD
ANDNOT 104.01  ; 左密封缸前进
OUT 104.02  ; 左密封缸后退
LD TR0
LD 161.01  ; 手动
AND 0.11  ; 接触器KM2辅助触点
AND 4.07  ; 排气孔密封缸向前
LD 161.00  ; 自动
AND 150.02  ; 输送线运行
AND 163.07  ; 排气孔密封缸前进
ORLD
ANDLD
LDNOT 3.12  ; 排气孔密封缸前位
ORNOT 3.10  ; 左密封缸前位
ANDLD
ANDNOT 104.04  ; 排气孔密封缸后退
OUT 104.03  ; 排气孔密封缸前进
LD TR0
LD 161.01  ; 手动
AND 0.11  ; 接触器KM2辅助触点
AND 4.08  ; 排气孔密封缸向后
LD 161.00  ; 自动
AND 150.02  ; 输送线运行
AND 163.08  ; 排气孔密封缸后退
ORLD
ANDLD
LDNOT 3.11  ; 排气孔密封缸后位
ORNOT 3.09  ; 左密封缸后位
ANDLD
ANDNOT 104.03  ; 排气孔密封缸前进
OUT 104.04  ; 排气孔密封缸后退
; rung 8
LDNOT 1.15  ; 品种选择
LD 161.01  ; 手动
AND 0.11  ; 接触器KM2辅助触点
AND 4.09  ; 工位停止器下
LD 161.00  ; 自动
AND 150.02  ; 输送线运行
AND 163.09  ; 工位停止器
ORLD
ANDLD
LD 1.15  ; 品种选择
LD 160.01  ; 手动
AND 0.11  ; 接触器KM2辅助触点
AND 4.09  ; 工位停止器下
LD 160.00  ; 自动
AND 150.02  ; 输送线运行
AND 163.09  ; 工位停止器
ORLD
ANDLD
ORLD
OUT 103.13  ; 工位停止器

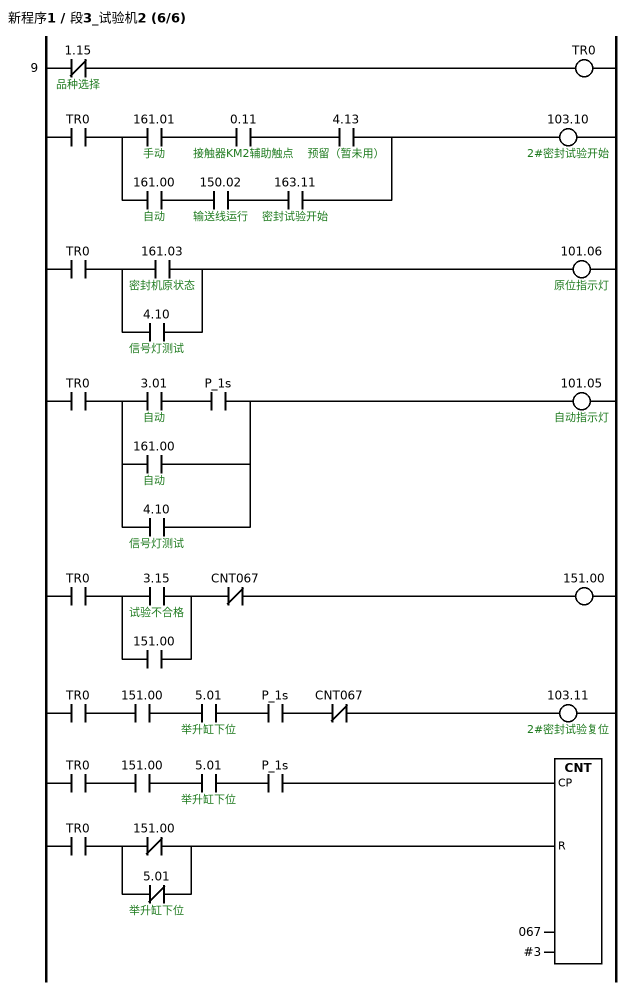
; rung 9
LDNOT 1.15  ; 品种选择
OUT TR0
LD 161.01  ; 手动
AND 0.11  ; 接触器KM2辅助触点
AND 4.13  ; 预留（暂未用）
LD 161.00  ; 自动
AND 150.02  ; 输送线运行
AND 163.11  ; 密封试验开始
ORLD
ANDLD
OUT 103.10  ; 2#密封试验开始
LD TR0
LD 161.03  ; 密封机原状态
OR 4.10  ; 信号灯测试
ANDLD
OUT 101.06  ; 原位指示灯
LD TR0
LD 3.01  ; 自动
AND P_1s
OR 161.00  ; 自动
OR 4.10  ; 信号灯测试
ANDLD
OUT 101.05  ; 自动指示灯
LD TR0
LD 3.15  ; 试验不合格
OR 151.00
ANDLD
ANDNOT CNT067
OUT 151.00
LD TR0
AND 151.00
AND 5.01  ; 举升缸下位
AND P_1s
ANDNOT CNT067
OUT 103.11  ; 2#密封试验复位
LD TR0
AND 151.00
AND 5.01  ; 举升缸下位
AND P_1s
LD TR0
LDNOT 151.00
ORNOT 5.01  ; 举升缸下位
ANDLD
CNT 067 #3

### Section 段4_维修段

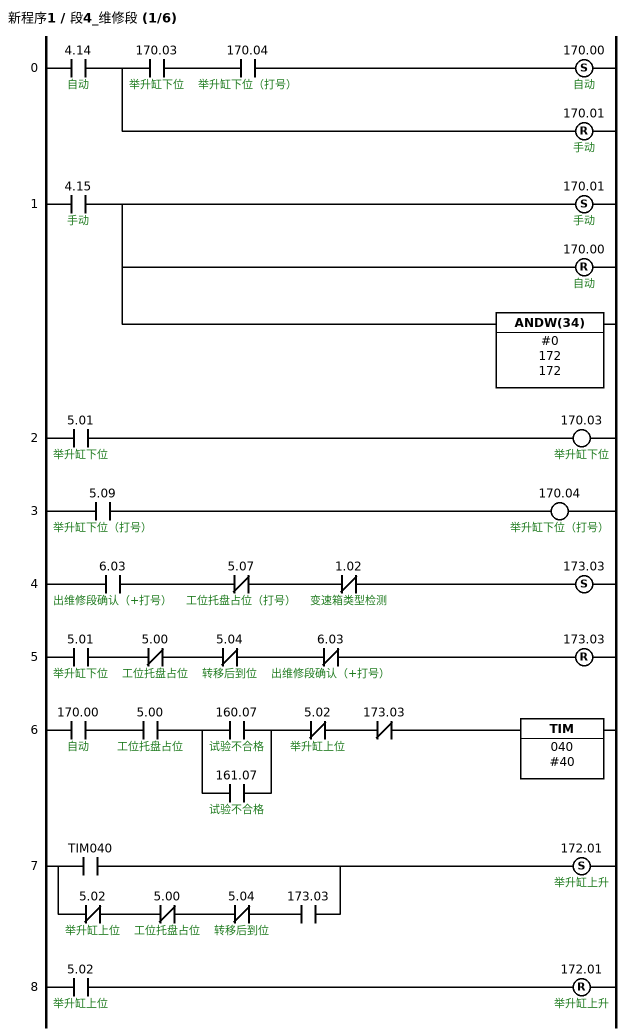
; rung 0
LD 4.14  ; 自动
OUT TR0
AND 170.03  ; 举升缸下位
AND 170.04  ; 举升缸下位（打号）
SET 170.00  ; 自动
LD TR0
RSET 170.01  ; 手动
; rung 1
LD 4.15  ; 手动
SET 170.01  ; 手动
RSET 170.00  ; 自动
ANDW(34) #0 172 172
; rung 2
LD 5.01  ; 举升缸下位
OUT 170.03  ; 举升缸下位
; rung 3
LD 5.09  ; 举升缸下位（打号）
OUT 170.04  ; 举升缸下位（打号）
; rung 4
LD 6.03  ; 出维修段确认（+打号）
ANDNOT 5.07  ; 工位托盘占位（打号）
ANDNOT 1.02  ; 变速箱类型检测
SET 173.03
; rung 5
LD 5.01  ; 举升缸下位
ANDNOT 5.00  ; 工位托盘占位
ANDNOT 5.04  ; 转移后到位
ANDNOT 6.03  ; 出维修段确认（+打号）
RSET 173.03
; rung 6
LD 170.00  ; 自动
AND 5.00  ; 工位托盘占位
LD 160.07  ; 试验不合格
OR 161.07  ; 试验不合格
ANDLD
ANDNOT 5.02  ; 举升缸上位
ANDNOT 173.03
TIM 040 #40
; rung 7
LD TIM040
LDNOT 5.02  ; 举升缸上位
ANDNOT 5.00  ; 工位托盘占位
ANDNOT 5.04  ; 转移后到位
AND 173.03
ORLD
SET 172.01  ; 举升缸上升
; rung 8
LD 5.02  ; 举升缸上位
RSET 172.01  ; 举升缸上升

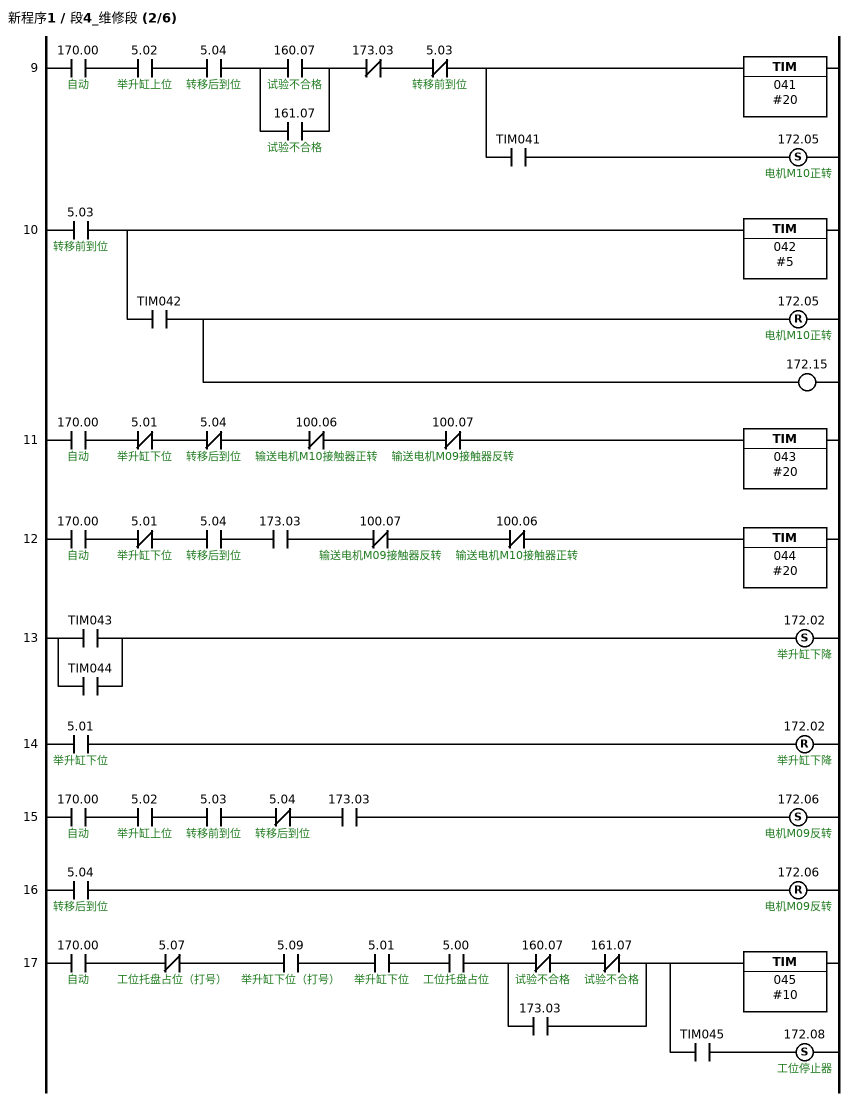
; rung 9
LD 170.00  ; 自动
AND 5.02  ; 举升缸上位
AND 5.04  ; 转移后到位
LD 160.07  ; 试验不合格
OR 161.07  ; 试验不合格
ANDLD
ANDNOT 173.03
ANDNOT 5.03  ; 转移前到位
TIM 041 #20
AND TIM041
SET 172.05  ; 电机M10正转
; rung 10
LD 5.03  ; 转移前到位
TIM 042 #5
AND TIM042
RSET 172.05  ; 电机M10正转
OUT 172.15
; rung 11
LD 170.00  ; 自动
ANDNOT 5.01  ; 举升缸下位
ANDNOT 5.04  ; 转移后到位
ANDNOT 100.06  ; 输送电机M10接触器正转
ANDNOT 100.07  ; 输送电机M09接触器反转
TIM 043 #20
; rung 12
LD 170.00  ; 自动
ANDNOT 5.01  ; 举升缸下位
AND 5.04  ; 转移后到位
AND 173.03
ANDNOT 100.07  ; 输送电机M09接触器反转
ANDNOT 100.06  ; 输送电机M10接触器正转
TIM 044 #20
; rung 13
LD TIM043
OR TIM044
SET 172.02  ; 举升缸下降
; rung 14
LD 5.01  ; 举升缸下位
RSET 172.02  ; 举升缸下降
; rung 15
LD 170.00  ; 自动
AND 5.02  ; 举升缸上位
AND 5.03  ; 转移前到位
ANDNOT 5.04  ; 转移后到位
AND 173.03
SET 172.06  ; 电机M09反转
; rung 16
LD 5.04  ; 转移后到位
RSET 172.06  ; 电机M09反转
; rung 17
LD 170.00  ; 自动
ANDNOT 5.07  ; 工位托盘占位（打号）
AND 5.09  ; 举升缸下位（打号）
AND 5.01  ; 举升缸下位
AND 5.00  ; 工位托盘占位
LDNOT 160.07  ; 试验不合格
ANDNOT 161.07  ; 试验不合格
OR 173.03
ANDLD
TIM 045 #10
AND TIM045
SET 172.08  ; 工位停止器

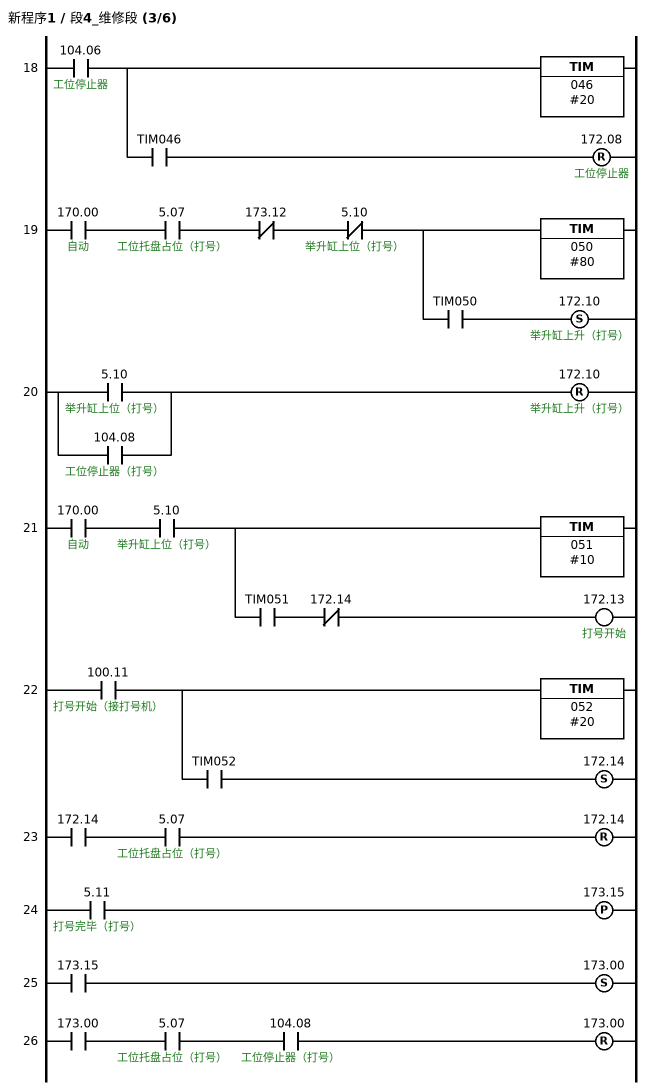
; rung 18
LD 104.06  ; 工位停止器
TIM 046 #20
AND TIM046
RSET 172.08  ; 工位停止器
; rung 19
LD 170.00  ; 自动
AND 5.07  ; 工位托盘占位（打号）
ANDNOT 173.12
ANDNOT 5.10  ; 举升缸上位（打号）
TIM 050 #80
AND TIM050
SET 172.10  ; 举升缸上升（打号）
; rung 20
LD 5.10  ; 举升缸上位（打号）
OR 104.08  ; 工位停止器（打号）
RSET 172.10  ; 举升缸上升（打号）
; rung 21
LD 170.00  ; 自动
AND 5.10  ; 举升缸上位（打号）
TIM 051 #10
AND TIM051
ANDNOT 172.14
OUT 172.13  ; 打号开始
; rung 22
LD 100.11  ; 打号开始（接打号机）
TIM 052 #20
AND TIM052
SET 172.14
; rung 23
LD 172.14
AND 5.07  ; 工位托盘占位（打号）
RSET 172.14
; rung 24
LD 5.11  ; 打号完毕（打号）
DIFU(13) 173.15
; rung 25
LD 173.15
SET 173.00
; rung 26
LD 173.00
AND 5.07  ; 工位托盘占位（打号）
AND 104.08  ; 工位停止器（打号）
RSET 173.00

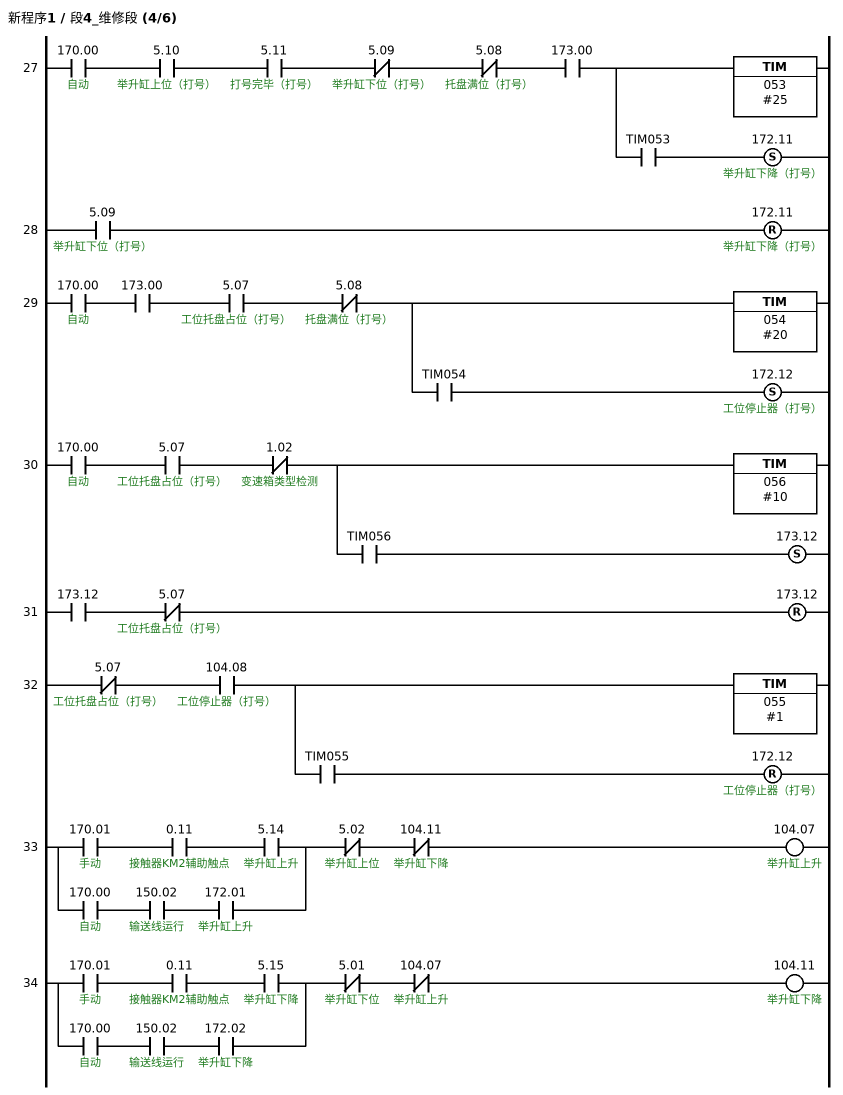
; rung 27
LD 170.00  ; 自动
AND 5.10  ; 举升缸上位（打号）
AND 5.11  ; 打号完毕（打号）
ANDNOT 5.09  ; 举升缸下位（打号）
ANDNOT 5.08  ; 托盘满位（打号）
AND 173.00
TIM 053 #25
AND TIM053
SET 172.11  ; 举升缸下降（打号）
; rung 28
LD 5.09  ; 举升缸下位（打号）
RSET 172.11  ; 举升缸下降（打号）
; rung 29
LD 170.00  ; 自动
AND 173.00
AND 5.07  ; 工位托盘占位（打号）
ANDNOT 5.08  ; 托盘满位（打号）
TIM 054 #20
AND TIM054
SET 172.12  ; 工位停止器（打号）
; rung 30
LD 170.00  ; 自动
AND 5.07  ; 工位托盘占位（打号）
ANDNOT 1.02  ; 变速箱类型检测
TIM 056 #10
AND TIM056
SET 173.12
; rung 31
LD 173.12
ANDNOT 5.07  ; 工位托盘占位（打号）
RSET 173.12
; rung 32
LDNOT 5.07  ; 工位托盘占位（打号）
AND 104.08  ; 工位停止器（打号）
TIM 055 #1
AND TIM055
RSET 172.12  ; 工位停止器（打号）
; rung 33
LD 170.01  ; 手动
AND 0.11  ; 接触器KM2辅助触点
AND 5.14  ; 举升缸上升
LD 170.00  ; 自动
AND 150.02  ; 输送线运行
AND 172.01  ; 举升缸上升
ORLD
ANDNOT 5.02  ; 举升缸上位
ANDNOT 104.11  ; 举升缸下降
OUT 104.07  ; 举升缸上升
; rung 34
LD 170.01  ; 手动
AND 0.11  ; 接触器KM2辅助触点
AND 5.15  ; 举升缸下降
LD 170.00  ; 自动
AND 150.02  ; 输送线运行
AND 172.02  ; 举升缸下降
ORLD
ANDNOT 5.01  ; 举升缸下位
ANDNOT 104.07  ; 举升缸上升
OUT 104.11  ; 举升缸下降

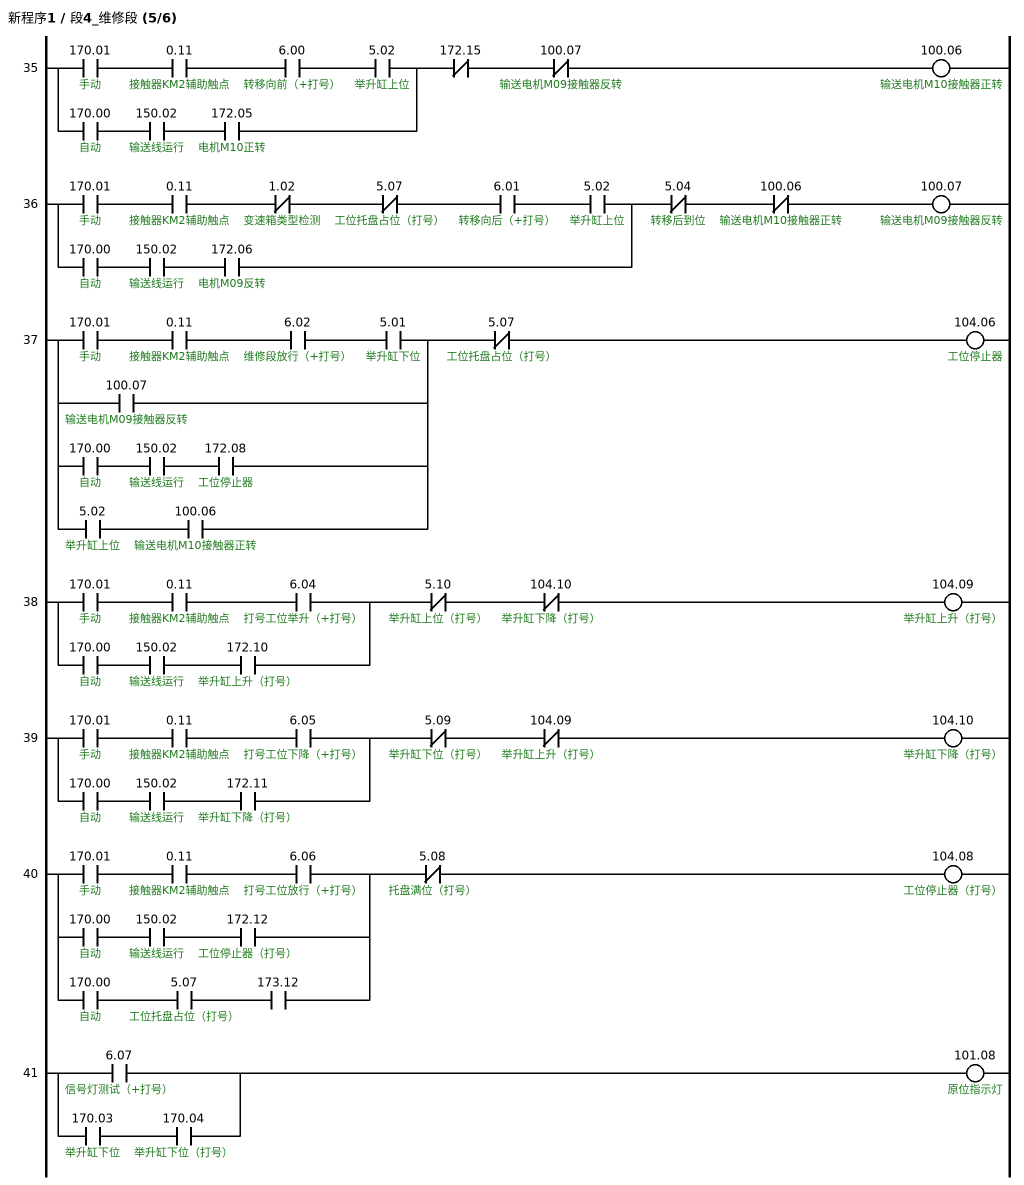
; rung 35
LD 170.01  ; 手动
AND 0.11  ; 接触器KM2辅助触点
AND 6.00  ; 转移向前（+打号）
AND 5.02  ; 举升缸上位
LD 170.00  ; 自动
AND 150.02  ; 输送线运行
AND 172.05  ; 电机M10正转
ORLD
ANDNOT 172.15
ANDNOT 100.07  ; 输送电机M09接触器反转
OUT 100.06  ; 输送电机M10接触器正转
; rung 36
LD 170.01  ; 手动
AND 0.11  ; 接触器KM2辅助触点
ANDNOT 1.02  ; 变速箱类型检测
ANDNOT 5.07  ; 工位托盘占位（打号）
AND 6.01  ; 转移向后（+打号）
AND 5.02  ; 举升缸上位
LD 170.00  ; 自动
AND 150.02  ; 输送线运行
AND 172.06  ; 电机M09反转
ORLD
ANDNOT 5.04  ; 转移后到位
ANDNOT 100.06  ; 输送电机M10接触器正转
OUT 100.07  ; 输送电机M09接触器反转
; rung 37
LD 170.01  ; 手动
AND 0.11  ; 接触器KM2辅助触点
AND 6.02  ; 维修段放行（+打号）
AND 5.01  ; 举升缸下位
OR 100.07  ; 输送电机M09接触器反转
LD 170.00  ; 自动
AND 150.02  ; 输送线运行
AND 172.08  ; 工位停止器
ORLD
LD 5.02  ; 举升缸上位
AND 100.06  ; 输送电机M10接触器正转
ORLD
ANDNOT 5.07  ; 工位托盘占位（打号）
OUT 104.06  ; 工位停止器
; rung 38
LD 170.01  ; 手动
AND 0.11  ; 接触器KM2辅助触点
AND 6.04  ; 打号工位举升（+打号）
LD 170.00  ; 自动
AND 150.02  ; 输送线运行
AND 172.10  ; 举升缸上升（打号）
ORLD
ANDNOT 5.10  ; 举升缸上位（打号）
ANDNOT 104.10  ; 举升缸下降（打号）
OUT 104.09  ; 举升缸上升（打号）
; rung 39
LD 170.01  ; 手动
AND 0.11  ; 接触器KM2辅助触点
AND 6.05  ; 打号工位下降（+打号）
LD 170.00  ; 自动
AND 150.02  ; 输送线运行
AND 172.11  ; 举升缸下降（打号）
ORLD
ANDNOT 5.09  ; 举升缸下位（打号）
ANDNOT 104.09  ; 举升缸上升（打号）
OUT 104.10  ; 举升缸下降（打号）
; rung 40
LD 170.01  ; 手动
AND 0.11  ; 接触器KM2辅助触点
AND 6.06  ; 打号工位放行（+打号）
LD 170.00  ; 自动
AND 150.02  ; 输送线运行
AND 172.12  ; 工位停止器（打号）
ORLD
LD 170.00  ; 自动
AND 5.07  ; 工位托盘占位（打号）
AND 173.12
ORLD
ANDNOT 5.08  ; 托盘满位（打号）
OUT 104.08  ; 工位停止器（打号）
; rung 41
LD 6.07  ; 信号灯测试（+打号）
LD 170.03  ; 举升缸下位
AND 170.04  ; 举升缸下位（打号）
ORLD
OUT 101.08  ; 原位指示灯

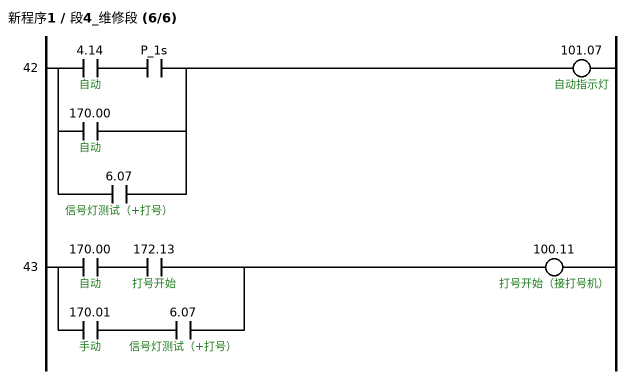
; rung 42
LD 4.14  ; 自动
AND P_1s
OR 170.00  ; 自动
OR 6.07  ; 信号灯测试（+打号）
OUT 101.07  ; 自动指示灯
; rung 43
LD 170.00  ; 自动
AND 172.13  ; 打号开始
LD 170.01  ; 手动
AND 6.07  ; 信号灯测试（+打号）
ORLD
OUT 100.11  ; 打号开始（接打号机）

### Section END
; rung 0
END(01)